TYPE TestSuiteHandle_t : POINTER TO FB_TestSuite; END_TYPE

(* stored: Version 1.1.0.1, ProductVersion 3.1.4022.9
   DUT TestSuiteHandle_t: Id {4c6be0e1-fd4b-4671-aeb6-cca131117c9d} *)
